INTERFACE IComparer EXTENDS IObject

METHOD Compare : COMPARISION_RESULT
VAR_INPUT
	left : GENERIC_VALUE;
	right : GENERIC_VALUE;
END_VAR
END_METHOD

END_INTERFACE

(* stored: Version 1.1.0.1
   Itf IComparer: Id {3b04600d-2a0c-4e89-8bfb-cd112c3ad567}
   Method Compare: Id {a0e4701a-7352-4984-98c4-52eaf1804d93} *)
